// TIA Portal V19 export
FUNCTION_BLOCK "DiesLubrication_FB"   // FB153, LAD
TITLE = DIES LUBRICATION
// stored: Access Published, MemoryReserve 100, SetENOAutomatically false
   VAR_INPUT
      AreaInterface : "AreaInterface";
      DataIn : Struct
         PbStop : Bool;
         PbStart : Bool;
         SensorLevel : Bool;
         ConnectorPlugged : Bool;
      END_STRUCT;
      CIn : Struct
         EnableStopInPhase : Bool;
         EnableStopProgrammed : Bool;
         EnableAborting : Bool;
         JobDone : Bool;
         ExternalPumpCycleDone : Bool;
         CutBenchCode : DInt;
      END_STRUCT;
      Config : Struct
         EnableWngSystemOff : Bool;
         ExternalPump : Bool;
         PumpWorkDuration : Time;
         PumpPauseDuration : Time;
         LowTankLevelDly : Time;
      END_STRUCT;
   END_VAR
   VAR_OUTPUT
      MachineInterface : "MachineInterface";
      DataOut : Struct
         PneumaticPumpSolenoidValve : Bool;
         Lamp : Bool;
      END_STRUCT;
      COut : Struct
         IsRunning : Bool;
         ToolsJobCounter : UDInt;
         PumpCycleCounter : UDInt;
      END_STRUCT;
   END_VAR
   VAR_IN_OUT
      PersistentValues : Struct
         Data : Struct
            SavedCutBenchCode : DInt;
            PumpJobCounter : UDInt;
            JobsCounter : UDInt;
         END_STRUCT;
         Par : Struct
            SystemOffOn : Bool;
            JobsToStart : UDInt;
            OilPumpCycles : UDInt;
         END_STRUCT;
      END_STRUCT;
   END_VAR
   VAR
      Sts : Struct
         AlarmsPresence : Bool;
         WarningsPresence : Bool;
         IsStandstill : Bool;
         PumpPauseDone : Bool;
         PumpWorkDone : Bool;
         LubNormCycleReq : Bool;
         Condition { ExternalAccessible := 'False'; ExternalVisible := 'False'; ExternalWritable := 'False'} : Bool;
      END_STRUCT;
      Ctrl : Struct
         RstAlarms : Bool;
         SafeMotion : Bool;
         StopDoorOpen : Bool;
         StopSafe : Bool;
         StopInPhase : Bool;
         StopProgrammed : Bool;
         ManStart : Bool;
         AutStart : Bool;
         V_Pneumatic : Bool;
      END_STRUCT;
      Warning : Struct
         NoAutReady : Bool;
         SystemOff : Bool;
      END_STRUCT;
      Alarm : Struct
         LowTankLevel : Bool;
         ConnectorUnplugged : Bool;
      END_STRUCT;
      TON_PumpPause : IEC_TIMER;
      TON_PumpWork : IEC_TIMER;
      TON_LowTankLevel : IEC_TIMER;
      JobDonePEAux : Bool;
      PbStartPEAux : Bool;
   END_VAR
   VAR_TEMP
      CutBechChanged : Bool;
      JobDonePositiveEdge : Bool;
   END_VAR
   VAR_TEMP   // added for the SCL form of the ladder/FBD networks
      _w1 : Bool;
      _w2 : Bool;
   END_VAR
BEGIN

REGION Network 1 (SCL): Reset alarms command
   #Ctrl.RstAlarms := #AreaInterface.RstAlarms;

   IF #Ctrl.RstAlarms THEN
       #Warning.NoAutReady := FALSE;
       #Alarm.LowTankLevel := FALSE;
       #Alarm.ConnectorUnplugged := FALSE;
   END_IF;
END_REGION

REGION Network 2: Warning system is off
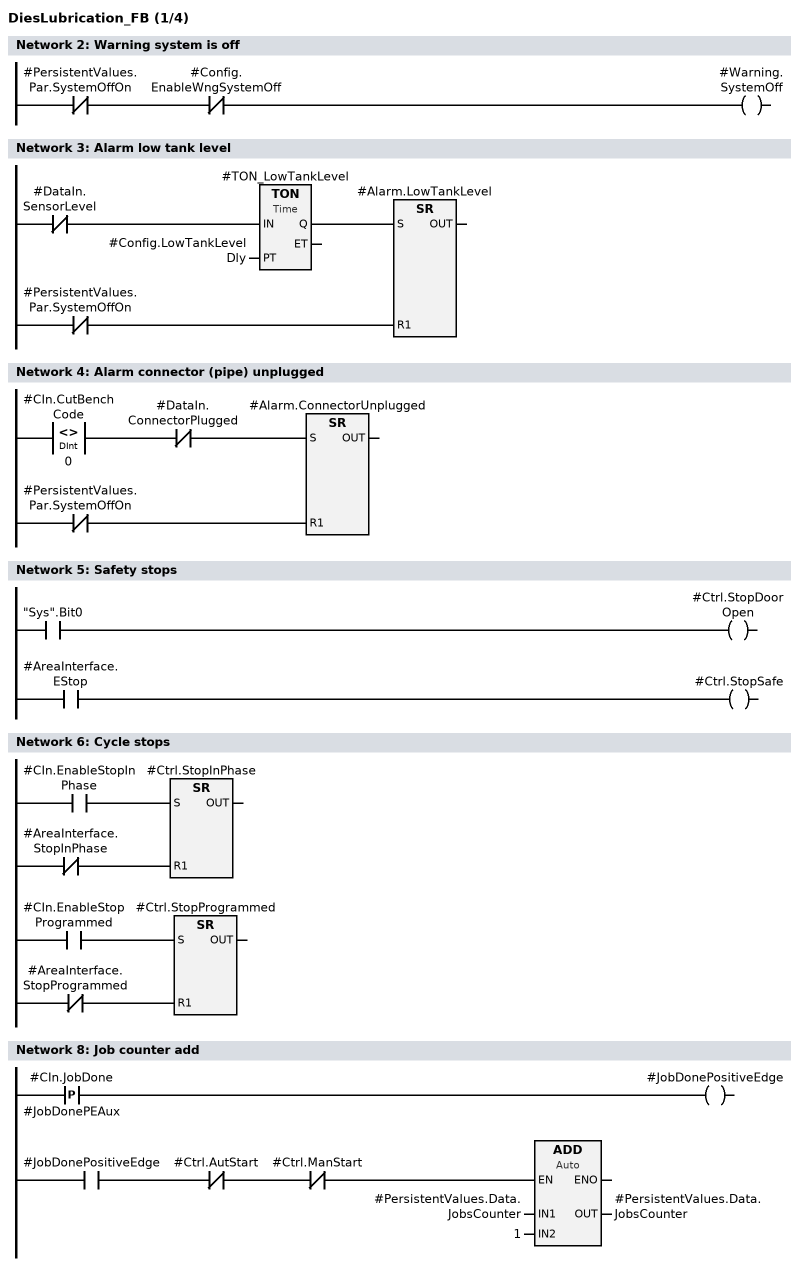
   RUNG wire#powerrail
      I_Contact( #PersistentValues.Par.SystemOffOn )
      I_Contact( #Config.EnableWngSystemOff )
      Coil( #Warning.SystemOff )
   END_RUNG
   // the same network as SCL:
   #Warning.SystemOff := NOT #PersistentValues.Par.SystemOffOn AND NOT #Config.EnableWngSystemOff;
END_REGION

REGION Network 3: Alarm low tank level
   RUNG wire#powerrail
      I_Contact( #DataIn.SensorLevel )
      { S7_Templates := "time_type := Time" } #TON_LowTankLevel.TON(pt := #Config.LowTankLevelDly, et =>)
      S_SR(operand := #Alarm.LowTankLevel, r1 := wire#w1)
   END_RUNG
   RUNG wire#powerrail
      I_Contact( #PersistentValues.Par.SystemOffOn )
   END_RUNG wire#w1
   // the same network as SCL:
   #TON_LowTankLevel.TON(IN := NOT #DataIn.SensorLevel, PT := #Config.LowTankLevelDly);
   IF #TON_LowTankLevel.Q THEN
       #Alarm.LowTankLevel := TRUE;   // SR flip-flop
   END_IF;
   IF NOT #PersistentValues.Par.SystemOffOn THEN #Alarm.LowTankLevel := FALSE; END_IF;
END_REGION

REGION Network 4: Alarm connector (pipe) unplugged
   RUNG wire#powerrail
      { S7_Templates := "SrcType := DInt" } NE_Contact(in1 := #CIn.CutBenchCode, in2 := 0)
      I_Contact( #DataIn.ConnectorPlugged )
      S_SR(operand := #Alarm.ConnectorUnplugged, r1 := wire#w1)
   END_RUNG
   RUNG wire#powerrail
      I_Contact( #PersistentValues.Par.SystemOffOn )
   END_RUNG wire#w1
   // the same network as SCL:
   IF (#CIn.CutBenchCode <> 0) AND NOT #DataIn.ConnectorPlugged THEN
       #Alarm.ConnectorUnplugged := TRUE;   // SR flip-flop
   END_IF;
   IF NOT #PersistentValues.Par.SystemOffOn THEN #Alarm.ConnectorUnplugged := FALSE; END_IF;
END_REGION

REGION Network 5: Safety stops
   RUNG wire#powerrail
      Contact( "Sys".Bit0 )
      Coil( #Ctrl.StopDoorOpen )
   END_RUNG
   RUNG wire#powerrail
      Contact( #AreaInterface.EStop )
      Coil( #Ctrl.StopSafe )
   END_RUNG
   // the same network as SCL:
   #Ctrl.StopDoorOpen := "Sys".Bit0;
   #Ctrl.StopSafe := #AreaInterface.EStop;
END_REGION

REGION Network 6: Cycle stops
   RUNG wire#powerrail
      Contact( #CIn.EnableStopInPhase )
      S_SR(operand := #Ctrl.StopInPhase, r1 := wire#w1)
   END_RUNG
   RUNG wire#powerrail
      I_Contact( #AreaInterface.StopInPhase )
   END_RUNG wire#w1
   RUNG wire#powerrail
      Contact( #CIn.EnableStopProgrammed )
      S_SR(operand := #Ctrl.StopProgrammed, r1 := wire#w2)
   END_RUNG
   RUNG wire#powerrail
      I_Contact( #AreaInterface.StopProgrammed )
   END_RUNG wire#w2
   // the same network as SCL:
   IF #CIn.EnableStopInPhase THEN
       #Ctrl.StopInPhase := TRUE;   // SR flip-flop
   END_IF;
   IF NOT #AreaInterface.StopInPhase THEN #Ctrl.StopInPhase := FALSE; END_IF;
   IF #CIn.EnableStopProgrammed THEN
       #Ctrl.StopProgrammed := TRUE;   // SR flip-flop
   END_IF;
   IF NOT #AreaInterface.StopProgrammed THEN #Ctrl.StopProgrammed := FALSE; END_IF;
END_REGION

REGION Network 7: <<< >>>
END_REGION

REGION Network 8: Job counter add
   RUNG wire#powerrail
      P_Contact(operand := #CIn.JobDone, bit := #JobDonePEAux)
      Coil( #JobDonePositiveEdge )
   END_RUNG
   RUNG wire#powerrail
      Contact( #JobDonePositiveEdge )
      I_Contact( #Ctrl.AutStart )
      I_Contact( #Ctrl.ManStart )
      Add(in1 := #PersistentValues.Data.JobsCounter, in2 := 1, out => #PersistentValues.Data.JobsCounter)
   END_RUNG
   // the same network as SCL:
   #_w1 := #CIn.JobDone AND NOT #JobDonePEAux;   // rising edge of #CIn.JobDone
   #JobDonePEAux := #CIn.JobDone;
   #JobDonePositiveEdge := #_w1;
   IF #JobDonePositiveEdge AND NOT #Ctrl.AutStart AND NOT #Ctrl.ManStart THEN
       #PersistentValues.Data.JobsCounter := #PersistentValues.Data.JobsCounter + 1;
   END_IF;
END_REGION

REGION Network 9: Cut bench code is change -> reset counters
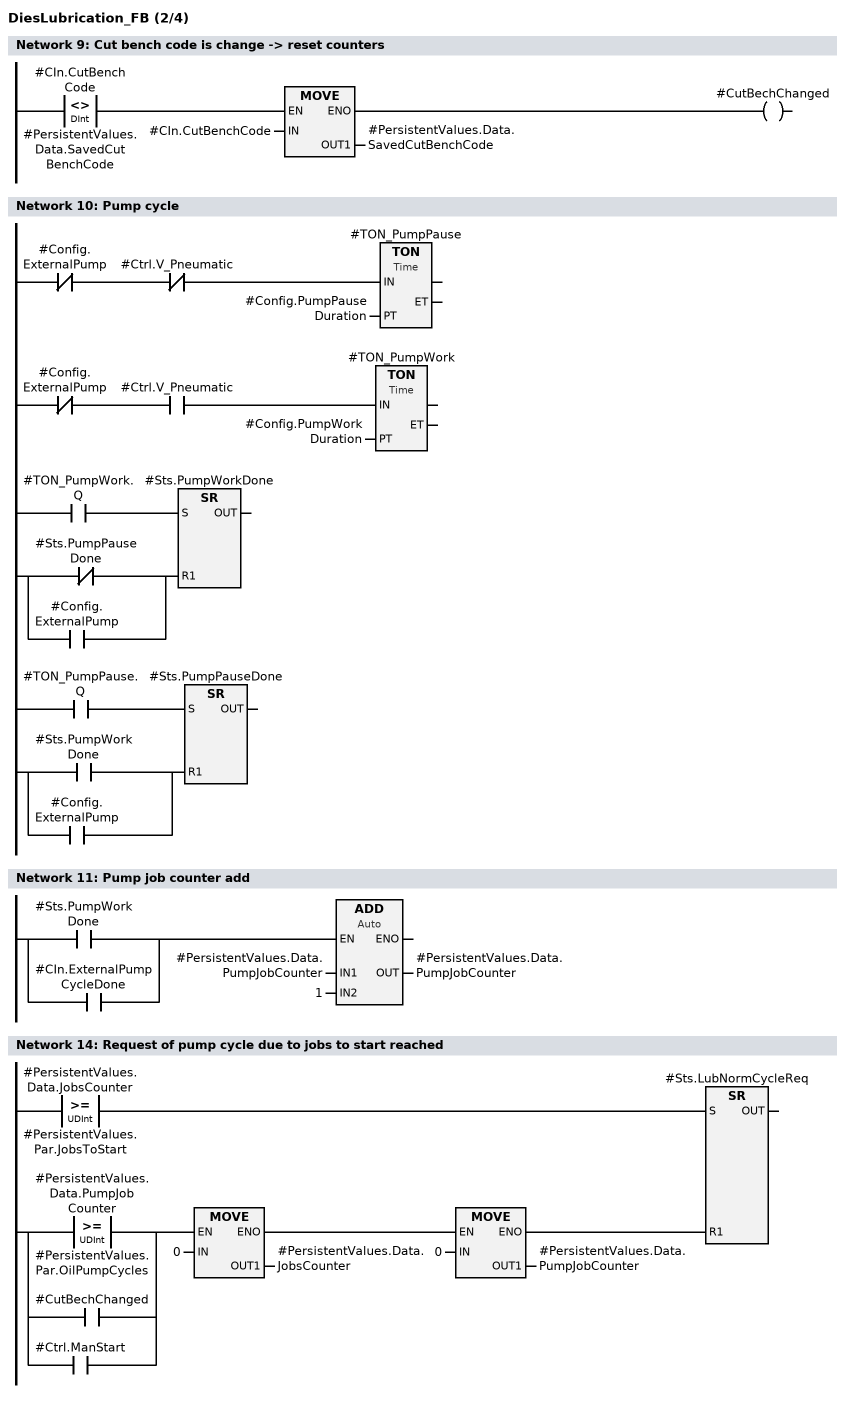
   RUNG wire#powerrail
      { S7_Templates := "SrcType := DInt" } NE_Contact(in1 := #CIn.CutBenchCode, in2 := #PersistentValues.Data.SavedCutBenchCode)
      Move(in := #CIn.CutBenchCode, out1 => #PersistentValues.Data.SavedCutBenchCode)
      Coil( #CutBechChanged )
   END_RUNG
   // the same network as SCL:
   #_w1 := #CIn.CutBenchCode <> #PersistentValues.Data.SavedCutBenchCode;
   IF #_w1 THEN #PersistentValues.Data.SavedCutBenchCode := #CIn.CutBenchCode; END_IF;
   #CutBechChanged := #_w1;
END_REGION

REGION Network 10: Pump cycle
   RUNG wire#powerrail
      I_Contact( #Config.ExternalPump )
      I_Contact( #Ctrl.V_Pneumatic )
      { S7_Templates := "time_type := Time" } #TON_PumpPause.TON(pt := #Config.PumpPauseDuration, et =>)
   END_RUNG
   RUNG wire#powerrail
      I_Contact( #Config.ExternalPump )
      Contact( #Ctrl.V_Pneumatic )
      { S7_Templates := "time_type := Time" } #TON_PumpWork.TON(pt := #Config.PumpWorkDuration, et =>)
   END_RUNG
   RUNG wire#powerrail
      Contact( #TON_PumpWork.Q )
      S_SR(operand := #Sts.PumpWorkDone, r1 := wire#w1)
   END_RUNG
   RUNG wire#powerrail
      I_Contact( #Sts.PumpPauseDone )
   END_RUNG wire#w1
   RUNG wire#powerrail
      Contact( #Config.ExternalPump )
   END_RUNG wire#w1
   RUNG wire#powerrail
      Contact( #TON_PumpPause.Q )
      S_SR(operand := #Sts.PumpPauseDone, r1 := wire#w2)
   END_RUNG
   RUNG wire#powerrail
      Contact( #Sts.PumpWorkDone )
   END_RUNG wire#w2
   RUNG wire#powerrail
      Contact( #Config.ExternalPump )
   END_RUNG wire#w2
   // the same network as SCL:
   #TON_PumpPause.TON(IN := NOT #Config.ExternalPump AND NOT #Ctrl.V_Pneumatic, PT := #Config.PumpPauseDuration);
   #TON_PumpWork.TON(IN := NOT #Config.ExternalPump AND #Ctrl.V_Pneumatic, PT := #Config.PumpWorkDuration);
   IF #TON_PumpWork.Q THEN
       #Sts.PumpWorkDone := TRUE;   // SR flip-flop
   END_IF;
   IF NOT #Sts.PumpPauseDone OR #Config.ExternalPump THEN #Sts.PumpWorkDone := FALSE; END_IF;
   IF #TON_PumpPause.Q THEN
       #Sts.PumpPauseDone := TRUE;   // SR flip-flop
   END_IF;
   IF #Sts.PumpWorkDone OR #Config.ExternalPump THEN #Sts.PumpPauseDone := FALSE; END_IF;
END_REGION

REGION Network 11: Pump job counter add
   RUNG wire#powerrail
      Contact( #Sts.PumpWorkDone )
      wire#w1
      Add(in1 := #PersistentValues.Data.PumpJobCounter, in2 := 1, out => #PersistentValues.Data.PumpJobCounter)
   END_RUNG
   RUNG wire#powerrail
      Contact( #CIn.ExternalPumpCycleDone )
   END_RUNG wire#w1
   // the same network as SCL:
   IF #Sts.PumpWorkDone OR #CIn.ExternalPumpCycleDone THEN
       #PersistentValues.Data.PumpJobCounter := #PersistentValues.Data.PumpJobCounter + 1;
   END_IF;
END_REGION

REGION Network 12: Pump work delayed
END_REGION

REGION Network 13: Pump phases mem
END_REGION

REGION Network 14: Request of pump cycle due to jobs to start reached
   RUNG wire#powerrail
      { S7_Templates := "SrcType := UDInt" } GE_Contact(in1 := #PersistentValues.Data.JobsCounter, in2 := #PersistentValues.Par.JobsToStart)
      S_SR(operand := #Sts.LubNormCycleReq, r1 := wire#w2)
   END_RUNG
   RUNG wire#powerrail
      { S7_Templates := "SrcType := UDInt" } GE_Contact(in1 := #PersistentValues.Data.PumpJobCounter, in2 := #PersistentValues.Par.OilPumpCycles)
      wire#w1
      Move(in := 0, out1 => #PersistentValues.Data.JobsCounter)
      Move(in := 0, out1 => #PersistentValues.Data.PumpJobCounter)
   END_RUNG wire#w2
   RUNG wire#powerrail
      Contact( #CutBechChanged )
   END_RUNG wire#w1
   RUNG wire#powerrail
      Contact( #Ctrl.ManStart )
   END_RUNG wire#w1
   // the same network as SCL:
   #_w1 := (#PersistentValues.Data.PumpJobCounter >= #PersistentValues.Par.OilPumpCycles) OR #CutBechChanged OR #Ctrl.ManStart;
   #_w2 := #PersistentValues.Data.JobsCounter >= #PersistentValues.Par.JobsToStart;
   IF #_w1 THEN
       #PersistentValues.Data.JobsCounter := 0;
       #PersistentValues.Data.PumpJobCounter := 0;
   END_IF;
   IF #_w2 THEN
       #Sts.LubNormCycleReq := TRUE;   // SR flip-flop
   END_IF;
   IF #_w1 THEN #Sts.LubNormCycleReq := FALSE; END_IF;
END_REGION

REGION Network 15: Run condition
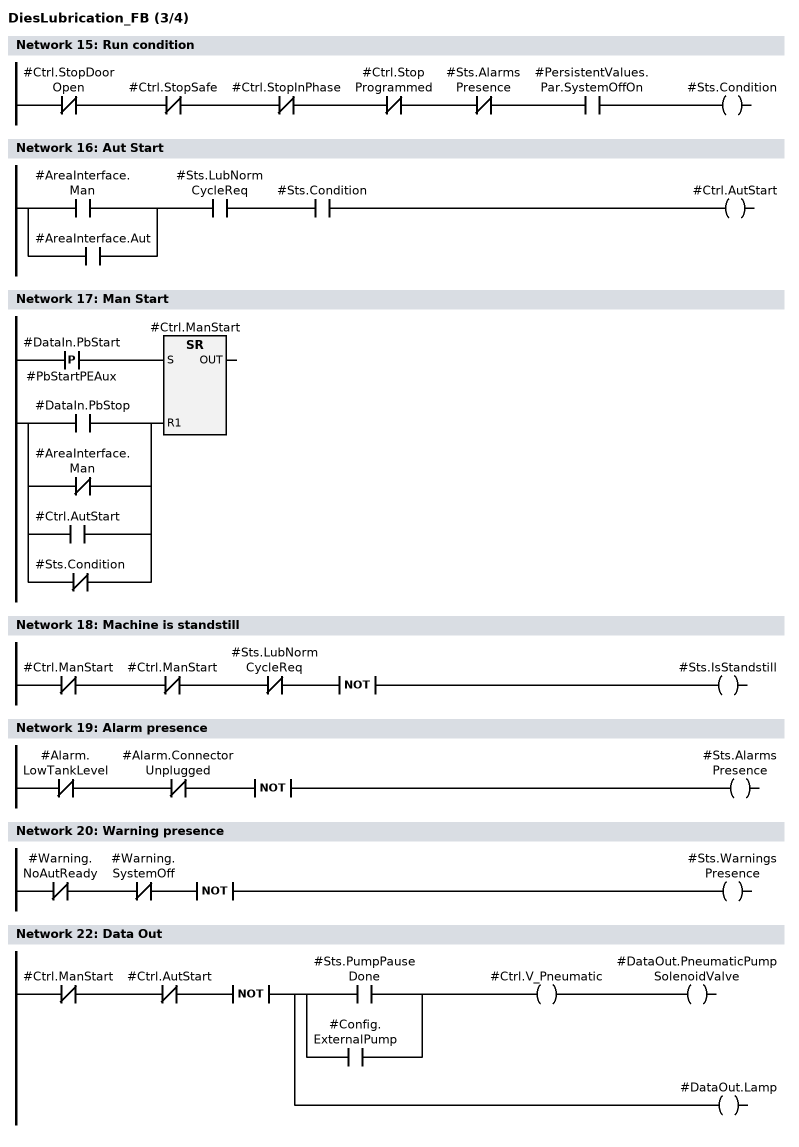
   RUNG wire#powerrail
      I_Contact( #Ctrl.StopDoorOpen )
      I_Contact( #Ctrl.StopSafe )
      I_Contact( #Ctrl.StopInPhase )
      I_Contact( #Ctrl.StopProgrammed )
      I_Contact( #Sts.AlarmsPresence )
      Contact( #PersistentValues.Par.SystemOffOn )
      Coil( #Sts.Condition )
   END_RUNG
   // the same network as SCL:
   #Sts.Condition := NOT #Ctrl.StopDoorOpen AND NOT #Ctrl.StopSafe AND NOT #Ctrl.StopInPhase AND NOT #Ctrl.StopProgrammed AND NOT #Sts.AlarmsPresence AND #PersistentValues.Par.SystemOffOn;
END_REGION

REGION Network 16: Aut Start
   RUNG wire#powerrail
      Contact( #AreaInterface.Man )
      wire#w1
      Contact( #Sts.LubNormCycleReq )
      Contact( #Sts.Condition )
      Coil( #Ctrl.AutStart )
   END_RUNG
   RUNG wire#powerrail
      Contact( #AreaInterface.Aut )
   END_RUNG wire#w1
   // the same network as SCL:
   #Ctrl.AutStart := (#AreaInterface.Man OR #AreaInterface.Aut) AND #Sts.LubNormCycleReq AND #Sts.Condition;
END_REGION

REGION Network 17: Man Start
   RUNG wire#powerrail
      P_Contact(operand := #DataIn.PbStart, bit := #PbStartPEAux)
      S_SR(operand := #Ctrl.ManStart, r1 := wire#w1)
   END_RUNG
   RUNG wire#powerrail
      Contact( #DataIn.PbStop )
   END_RUNG wire#w1
   RUNG wire#powerrail
      I_Contact( #AreaInterface.Man )
   END_RUNG wire#w1
   RUNG wire#powerrail
      Contact( #Ctrl.AutStart )
   END_RUNG wire#w1
   RUNG wire#powerrail
      I_Contact( #Sts.Condition )
   END_RUNG wire#w1
   // the same network as SCL:
   #_w1 := #DataIn.PbStart AND NOT #PbStartPEAux;   // rising edge of #DataIn.PbStart
   #PbStartPEAux := #DataIn.PbStart;
   IF #_w1 THEN
       #Ctrl.ManStart := TRUE;   // SR flip-flop
   END_IF;
   IF #DataIn.PbStop OR NOT #AreaInterface.Man OR #Ctrl.AutStart OR NOT #Sts.Condition THEN
       #Ctrl.ManStart := FALSE;
   END_IF;
END_REGION

REGION Network 18: Machine is standstill
   RUNG wire#powerrail
      I_Contact( #Ctrl.ManStart )
      I_Contact( #Ctrl.ManStart )
      I_Contact( #Sts.LubNormCycleReq )
      Not()
      Coil( #Sts.IsStandstill )
   END_RUNG
   // the same network as SCL:
   #Sts.IsStandstill := NOT (NOT #Ctrl.ManStart AND NOT #Ctrl.ManStart AND NOT #Sts.LubNormCycleReq);
END_REGION

REGION Network 19: Alarm presence
   RUNG wire#powerrail
      I_Contact( #Alarm.LowTankLevel )
      I_Contact( #Alarm.ConnectorUnplugged )
      Not()
      Coil( #Sts.AlarmsPresence )
   END_RUNG
   // the same network as SCL:
   #Sts.AlarmsPresence := NOT (NOT #Alarm.LowTankLevel AND NOT #Alarm.ConnectorUnplugged);
END_REGION

REGION Network 20: Warning presence
   RUNG wire#powerrail
      I_Contact( #Warning.NoAutReady )
      I_Contact( #Warning.SystemOff )
      Not()
      Coil( #Sts.WarningsPresence )
   END_RUNG
   // the same network as SCL:
   #Sts.WarningsPresence := NOT (NOT #Warning.NoAutReady AND NOT #Warning.SystemOff);
END_REGION

REGION Network 21 (SCL): Collect machine to area interface
   // Status machine ready
   #MachineInterface.AutReady := #AreaInterface.Aut AND NOT #Sts.AlarmsPresence;
   // Status machine aborting
   #MachineInterface.Aborting := #Sts.AlarmsPresence;
   // Status Ack Stop in phase
   #MachineInterface.AckStopInPhase := #Ctrl.StopInPhase;
   // Status Ack Stop programmed
   #MachineInterface.AckStopProgrammed := #Ctrl.StopProgrammed ;
   // Status Motion standtill
   #MachineInterface.MotionsStandStill := #Sts.IsStandstill;
   // Status Alarm presence
   #MachineInterface.AlarmsPresence := #Sts.AlarmsPresence;
   // Status Warning presence
   #MachineInterface.WarningPresence := #Sts.WarningsPresence;

   // Warning machine not automatic ready
   IF #AreaInterface.CheckAutReady AND NOT #MachineInterface.AutReady THEN
     #Warning.NoAutReady := TRUE;
   END_IF;
END_REGION

REGION Network 22: Data Out
   RUNG wire#powerrail
      I_Contact( #Ctrl.ManStart )
      I_Contact( #Ctrl.AutStart )
      Not()
      wire#w1
      Contact( #Sts.PumpPauseDone )
      wire#w2
      Coil( #Ctrl.V_Pneumatic )
      Coil( #DataOut.PneumaticPumpSolenoidValve )
   END_RUNG
   RUNG wire#w1
      Contact( #Config.ExternalPump )
   END_RUNG wire#w2
   RUNG wire#w1
      Coil( #DataOut.Lamp )
   END_RUNG
   // the same network as SCL:
   #_w1 := NOT (NOT #Ctrl.ManStart AND NOT #Ctrl.AutStart);
   #Ctrl.V_Pneumatic := #_w1 AND (#Sts.PumpPauseDone OR #Config.ExternalPump);
   #DataOut.PneumaticPumpSolenoidValve := #Ctrl.V_Pneumatic;
   #DataOut.Lamp := #_w1;
END_REGION

REGION Network 23: Coordination Out
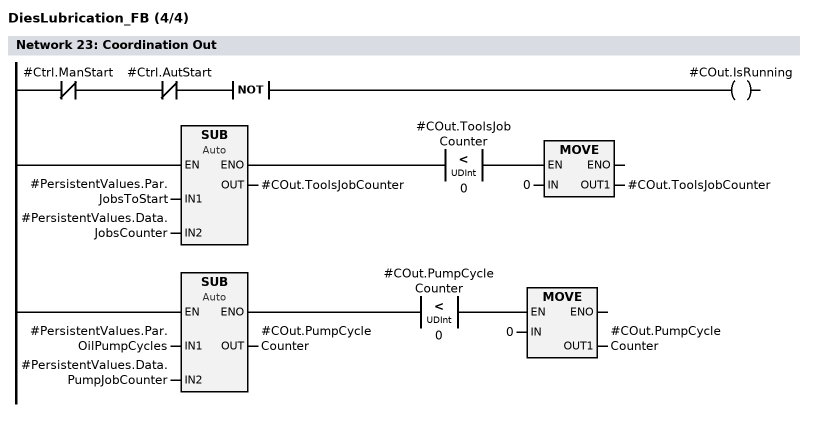
   RUNG wire#powerrail
      I_Contact( #Ctrl.ManStart )
      I_Contact( #Ctrl.AutStart )
      Not()
      Coil( #COut.IsRunning )
   END_RUNG
   RUNG wire#powerrail
      Sub(in1 := #PersistentValues.Par.JobsToStart, in2 := #PersistentValues.Data.JobsCounter, out => #COut.ToolsJobCounter)
      { S7_Templates := "SrcType := UDInt" } LT_Contact(in1 := #COut.ToolsJobCounter, in2 := 0)
      Move(in := 0, out1 => #COut.ToolsJobCounter)
   END_RUNG
   RUNG wire#powerrail
      Sub(in1 := #PersistentValues.Par.OilPumpCycles, in2 := #PersistentValues.Data.PumpJobCounter, out => #COut.PumpCycleCounter)
      { S7_Templates := "SrcType := UDInt" } LT_Contact(in1 := #COut.PumpCycleCounter, in2 := 0)
      Move(in := 0, out1 => #COut.PumpCycleCounter)
   END_RUNG
   // the same network as SCL:
   #COut.IsRunning := NOT (NOT #Ctrl.ManStart AND NOT #Ctrl.AutStart);
   #COut.ToolsJobCounter := #PersistentValues.Par.JobsToStart - #PersistentValues.Data.JobsCounter;
   IF #COut.ToolsJobCounter < 0 THEN #COut.ToolsJobCounter := 0; END_IF;
   #COut.PumpCycleCounter := #PersistentValues.Par.OilPumpCycles - #PersistentValues.Data.PumpJobCounter;
   IF #COut.PumpCycleCounter < 0 THEN #COut.PumpCycleCounter := 0; END_IF;
END_REGION
END_FUNCTION_BLOCK
